// TIA Portal V18 export
// export: Created 2026-01-09T11:23:39.007806Z, ExportSetting WithDefaults, DisplayName Totally Integrated Automation Portal, DisplayVersion V18 Update 5, DisplayName TIA Portal Openness, DisplayVersion V18 Update 5, DisplayName TIA Portal Teamcenter Gateway, DisplayVersion V18, DisplayName TIA Portal Version Control Interface, DisplayVersion V18, DisplayName SINAMICS Startdrive Advanced, DisplayVersion V18 SP2 Update 1, DisplayName SINAMICS Startdrive G110M, G120, G120C, G120D, G120P, G115D, DisplayVersion V18 SP2 Update 1, DisplayName SINAMICS Startdrive G130, G150, S120, S150, SINAMICS MV, S210, G220, S200, DisplayVersion V18 SP2 Update 1, DisplayName STEP 7 Professional, DisplayVersion V18 Update 5, DisplayName STEP 7 Safety, DisplayVersion V18, DisplayName WinCC Professional, DisplayVersion V18 Update 5
Screen "910MES_Com"  1280x800, Number=910, Template=09MES
  ScreenLayer 
    Rectangle "矩形_1" at 404,80 size 396x264  StyleItem=RectangleBackGD1
    Rectangle "矩形_2" at 0,80 size 396x320  StyleItem=RectangleBackGD1
  ScreenLayer 
    TextField "文本域_45" at 8,108 size 124x16  StyleItem=TxtMiddle24, Text="P-HeartBeat"
    SymbolicIOField "符号 I/O 域_1" at 136,108 size 132x16  CountVisibleItems=2, Mode=Output, OnValue=1, TextList=W-Heartbeat, TextOff="0", TextOn="1"
    TextField "文本域_8" at 0,80 size 360x24  Text="PLC TO MES - Common"
    TextField "文本域_7" at 408,126 size 124x16  StyleItem=TxtMiddle24, Text="M-HeartBeat"
    SymbolicIOField "符号 I/O 域_13" at 536,126 size 132x16  CountVisibleItems=2, Mode=Output, OnValue=1, TextList=W-Heartbeat, TextOff="0", TextOn="1"
    TextField "文本域_12" at 404,80 size 360x24  Text="MES TO PLC - Common"
